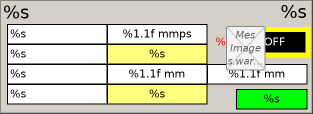
VISUALIZATION VISU_AXE_STD1_LIN_REL  // 313x114
VAR_IN_OUT
	m_Input_MOTEUR: BLOCK_AXE_STD1;
	m_Input_PRG_MOUVEMENT_PS: BLOCK_PRG_MOUVEMENT_PS;
END_VAR
VAR_Input
	m_Input_ID_NOM_XML : INT;
	m_Input_INDEX_MOTEUR : INT;
	m_Input_Ref_Trf:	INT;
	m_Input_NumFrame_Manu:	USINT;		(*numéro de frame à afficher dans le synoptique MANUEL*)
END_VAR
    Rectangle (0,0 313x114), "%s", text list: 'TextList_Type_Moteur', text index: m_Input_ID_NOM_XML
    Rectangle (223,4 87x16), "%s", text variable: m_Input_MOTEUR.MNEMO
    RoundedRectangle (7,24 100x20), "%s", text list: 'TextList_Moteurs', text index: 7
    RoundedRectangle (7,44 100x20), "%s", text list: 'TextList_Moteurs', text index: 8
    RoundedRectangle (7,64 100x20), "%s", text list: 'TextList_Moteurs', text index: 9
    RoundedRectangle (7,84 100x20), "%s", text list: 'TextList_Moteurs', text index: 10
    RoundedRectangle (107,24 100x20), "%1.1f mmps", text variable: m_Input_MOTEUR.STATE_Vit
    RoundedRectangle (107,44 100x20), "%s", text variable: m_Input_MOTEUR.CONF_ID_POSTE[m_Input_MOTEUR.PRM_NPOSTE]
    RoundedRectangle (107,64 100x20), "%1.1f mm", text variable: m_Input_MOTEUR.STATE_Pos_Rel
    RoundedRectangle (207,64 100x20), "%1.1f mm", text variable: m_Input_MOTEUR.STATE_Pos
    RoundedRectangle (107,84 100x20), "%s", text variable: m_Input_MOTEUR.CONF_ID_REF[m_Input_MOTEUR.PRM_NRef]
    RoundedRectangle (236,89 71x20), "%s", invisible if: m_Input_MOTEUR.STATE_Homed OR m_Input_MOTEUR.CONF_No_Ref, text list: 'TextList_Moteurs', text index: 11
    RoundedRectangle (236,89 71x20), "%s", invisible if: NOT m_Input_MOTEUR.STATE_Homed OR m_Input_MOTEUR.CONF_No_Ref, text list: 'TextList_Moteurs', text index: 11
    RoundedRectangle (240,27 70x30), invisible if: NOT m_Input_MOTEUR.OP_Validation.OK
    RoundedRectangle (240,27 70x30), invisible if: NOT m_Input_MOTEUR.OP_Validation.AR
    RoundedRectangle (240,27 70x30), invisible if: NOT m_Input_MOTEUR.OP_Validation.EC
    RoundedRectangle (245,32 60x20), "ON", invisible if: m_Input_MOTEUR.STATE_Ar
    RoundedRectangle (245,32 60x20), "OFF", invisible if: NOT m_Input_MOTEUR.STATE_Ar
    Rectangle (165,34 67x21), "%i", text variable: m_Input_MOTEUR.STATE_Err, invisible if: NOT m_Input_MOTEUR.STATE_NOK
    Image (226,26 39x44), invisible if: NOT m_Input_MOTEUR.STATE_NOK, image: MesImages.warning
    Rectangle (0,0 313x114)
        OnMouseClick: execute { .VISU_INDEX_MANU := m_Input_NumFrame_Manu; }
        OnMouseClick: change screen: SYN_MANUEL
END_VISUALIZATION

(* stored: Version 1.1.0.1, ProductVersion 3.1.4024.10
   Visu VISU_AXE_STD1_LIN_REL: Id {3e7502b8-71c8-4557-8723-fe78a1f62592} *)
